FUNCTION_BLOCK BasicBlock
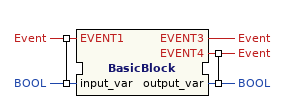
  EVENT_INPUT
    EVENT1 WITH input_var;
  END_EVENT
  EVENT_OUTPUT
    EVENT3;
    EVENT4 WITH output_var;
  END_EVENT
  VAR_INPUT
    input_var : BOOL;
  END_VAR
  VAR_OUTPUT
    output_var : BOOL;
  END_VAR
  EC_STATES
    START;
  END_STATES
END_FUNCTION_BLOCK
